(* IEC 61131-3 sources: std_i2980_v2.06_cp053/Source/IMM/ieccontrol/PumpGeneral, 8 files *)

(* ---- ABMeasure.pu ---- *)
(*
@h    ! WARNING !
@h    The Kemro K2 system (including software) only meets category B according to EN 954-1,
@h    thus it is not intended for usage in safety-relevant control applications in the field
@h    of personal safety (e.g. emergency stop).
@h    To implement potentially necessary safety-relevant control tasks, always use additional
@h    external safety devices that are intended for the particular purpose, and meet the necessary
@h    functional safety.
@h    For further information see EN 954-1 (EN ISO 13849-1) and/or the K2-x00 user manual, chapter
@h    "CE conformity, directives and standards".
*)

IMPORT_OVER_LISTFILE
 KAPPL_LintabData_2P
, KAPPL_MeasureMonitoring
, KSWO_Status
, ABMeasureAI

END_IMPORT

ALGORITHM_BLOCK ABMeasure #DUMMY_EDIT_BLOCK

SYSTEM_VAR
 sv_rActPressureHydr : REAL (* actual pressure in bar (measured by pressure sensor) *);
 ai_SysPressure : REAL;
 sv_SysPressureLintab : KAPPL_LintabData_2P (* lintab for measurement of system pressure sensor *);
 sv_SysPresMonitorMeas : KAPPL_MeasureMonitoring;
 sv_bDeviceReady : BOOL;
END_VAR

SYSTEM_OBJECT
 TaskInject : TASK;
 TaskSlow : TASK;
END_OBJECT

PROCESS_ALGORITHM paInitDebugMeasurement ON TaskSlow AUTOSTART

VAR
 variableName : STRING(255);
 swoState : KSWO_Status;
END_VAR
#BEGIN_EDIT_BLOCK
(**************************************** WARNING ********************************************
 *** The KEBA Kemro K2 System including software is not intended for safety control tasks! ***
 ***                       For further information see Comment tab!                        ***
 *********************************************************************************************)

variableName := CONCAT(GET_MY_FU_NAME(),'.sv_rActPressureHydr');
swoState := KSWO_AddVariable( Task := TaskInject,
                              Name := variableName,
                              Variable := sv_rActPressureHydr);

STOP_PROCESS_ALGORITHM();

;#END_EDIT_BLOCK END_ALGORITHM

PROCESS_ALGORITHM paMeasurePressure ON TaskInject(1000) AUTOSTART

VAR_TEMP
 b : BOOL;
END_VAR

VAR
 abPressureMeasure : ABMeasureAI;
 bSensorLinked : BOOL;
 sEndPoint : STRING(64);
END_VAR

(* IecGraph-Code *)

(* init step *)
INITIAL_STEP S_Start:
ACheckSensor (P);
END_STEP

ACTION ACheckSensor: #BEGIN_EDIT_BLOCK
bSensorLinked := IS_LINKED(ai_SysPressure);

;#END_EDIT_BLOCK END_ACTION (*ACheckSensor*)

(* steps *)
STEP S_Stop:
AStop (P);
END_STEP

ACTION AStop: #BEGIN_EDIT_BLOCK
STOP_PROCESS_ALGORITHM();

;#END_EDIT_BLOCK END_ACTION (*AStop*)
STEP S_Init:
AInitMeasure (P);
END_STEP

STEP S_Measure:
AMeasure (N);
END_STEP

(* transitions *)
TRANSITION TLinked (* TLinked *) FROM S_Start TO S_Init :=  #BEGIN_EDIT_BLOCK
bSensorLinked
;#END_EDIT_BLOCK
END_TRANSITION

TRANSITION TNotLinked (* TNotLinked *) FROM S_Start TO S_Stop :=  #BEGIN_EDIT_BLOCK
NOT bSensorLinked
;#END_EDIT_BLOCK
END_TRANSITION

TRANSITION TStop (* TStop *) FROM S_Stop TO S_Start :=  #BEGIN_EDIT_BLOCK
TRUE
;#END_EDIT_BLOCK
END_TRANSITION

TRANSITION TInitDone (* TInitDone *) FROM S_Init TO S_Measure :=  #BEGIN_EDIT_BLOCK
TRUE
;#END_EDIT_BLOCK
END_TRANSITION

(* end IecGraph-Code *)
(* sfc-code *)

(* stand alone actions *)
ACTION AInitMeasure: #BEGIN_EDIT_BLOCK
(**************************************** WARNING ********************************************
 *** The KEBA Kemro K2 System including software is not intended for safety control tasks! ***
 ***                       For further information see Comment tab!                        ***
 *********************************************************************************************)

sEndPoint := CONCAT(GET_MY_FU_NAME(),".ai_SysPressure");

abPressureMeasure.aInit(sRawValue:= sEndPoint,
                        pLintabPointArray := @sv_SysPressureLintab.LintabPoints.Point,
                        piUsedLintabPoints := @sv_SysPressureLintab.LintabPoints.uNoOfPoints);

abPressureMeasure.aInitMonitoring(bEnable := sv_SysPresMonitorMeas.EnableMonitoring,
                                  rLowLimit := sv_SysPresMonitorMeas.LowerLimit,
                                  bLimitation := sv_SysPresMonitorMeas.Limitation,
                                  rFailureFactor := sv_SysPresMonitorMeas.FailureFactor);

;#END_EDIT_BLOCK END_ACTION (*AInitMeasure*)
ACTION AMeasure: #BEGIN_EDIT_BLOCK
(**************************************** WARNING ********************************************
 *** The KEBA Kemro K2 System including software is not intended for safety control tasks! ***
 ***                       For further information see Comment tab!                        ***
 *********************************************************************************************)

abPressureMeasure.aRunLight(bIdle := sv_bDeviceReady);

b := WRITE_SVREAL_DIRECT(sv_rActPressureHydr, abPressureMeasure.aRunLight.rValue);

;#END_EDIT_BLOCK END_ACTION (*AMeasure*)
(* end sfc-code *)

END_ALGORITHM

END_ALGORITHM_BLOCK

#END_OF_IEC_PART

@Puma @IecEditor 6 149 @Pou 25
@@@BEG_Comment@@@
@h    ! WARNING !
@h    The Kemro K2 system (including software) only meets category B according to EN 954-1,
@h    thus it is not intended for usage in safety-relevant control applications in the field
@h    of personal safety (e.g. emergency stop).
@h    To implement potentially necessary safety-relevant control tasks, always use additional
@h    external safety devices that are intended for the particular purpose, and meet the necessary
@h    functional safety.
@h    For further information see EN 954-1 (EN ISO 13849-1) and/or the K2-x00 user manual, chapter
@h    "CE conformity, directives and standards".
@@@END_Comment@@@

@BEG_Contents

@BEG_Func
@RT(17)FuncTreeContainer
0
@END_Func

@BEG_Const
@RT(18)ConstTreeContainer
0
@END_Const

@BEG_Export

@BEG_Kind
@ALGORITHM_BLOCK @RT(9)ABMeasure @STRUCTURED_TEXT
@RT(0) @RT(0) @RT(0)
@END_Kind

@BEG_Dcl
@RT(16)DclTreeContainer
7
@Var @RT(10)TaskInject @RT(0) @T @T @RENAMED 0 @T @T @DT @RT(4)TASK @RT(0) @T @T @BASIC 0 @F
@F @F
@T
@BEG_Attrib
3 @RT(0) @RT(0) @RT(0)
@END_Attrib
1 7 @F @F @F @F

@Var @RT(8)TaskSlow @RT(0) @T @T @RENAMED 0 @T @T @DT @RT(4)TASK @RT(0) @T @T @BASIC 0 @F
@F @F
@T
@BEG_Attrib
3 @RT(0) @RT(0) @RT(0)
@END_Attrib
1 7 @F @F @F @F

@Var @RT(19)sv_rActPressureHydr @RT(0) @T @F @DT @RT(4)REAL @RT(0) @T @T @BASIC 0 @F
@F @F
@T
@BEG_Attrib
3 @RT(0) @RT(52)actual pressure in bar (measured by pressure sensor) @RT(0)
@END_Attrib
1 8 @F @F @F @F

@Var @RT(14)ai_SysPressure @RT(0) @T @F @DT @RT(4)REAL @RT(0) @T @T @BASIC 0 @F
@F @F
@T
@BEG_Attrib
3 @RT(0) @RT(0) @RT(0)
@END_Attrib
1 8 @F @F @F @F

@Var @RT(20)sv_SysPressureLintab @RT(0) @T @T @DERIVED 0 @F @RT(19)KAPPL_LintabData_2P @F
@T
@BEG_Attrib
3 @RT(0) @RT(48)lintab for measurement of system pressure sensor @RT(0)
@END_Attrib
1 8 @F @F @F @F

@Var @RT(21)sv_SysPresMonitorMeas @RT(0) @T @T @DERIVED 0 @T @T @DT @RT(23)KAPPL_MeasureMonitoring @RT(0) @T @T @UNKNOWN 0 @F
@F @F
@T
@BEG_Attrib
3 @RT(0) @RT(0) @RT(0)
@END_Attrib
1 8 @F @F @F @F

@Var @RT(15)sv_bDeviceReady @RT(0) @T @F @DT @RT(4)BOOL @RT(0) @T @T @BASIC 0 @F
@F @F
@T
@BEG_Attrib
3 @RT(0) @RT(0) @RT(0)
@END_Attrib
1 8 @F @F @F @F

@END_Dcl

@END_Export

@BEG_Body

2

@BEG_Export

@BEG_Algo
@PROCESS_ALGORITHM @RT(22)paInitDebugMeasurement @STRUCTURED_TEXT
@RT(0) @RT(0) @RT(8)TaskSlow @T @F
@END_Algo

@BEG_Dcl
@RT(16)DclTreeContainer
2
@Var @RT(12)variableName @RT(0) @T @F @DT @RT(11)STRING(255) @RT(0) @T @T @STRING 0 @F @RT(3)255 @F
@F @F
@T
@BEG_Attrib
3 @RT(0) @RT(0) @RT(0)
@END_Attrib
1 0 @F @F @F @F

@Var @RT(8)swoState @RT(0) @T @T @DERIVED 0 @T @T @DT @RT(11)KSWO_Status @RT(0) @T @T @UNKNOWN 0 @F
@F @F
@T
@BEG_Attrib
3 @RT(0) @RT(0) @RT(0)
@END_Attrib
1 0 @F @F @F @F

@END_Dcl

@END_Export

@BEG_Export

@BEG_Algo
@PROCESS_ALGORITHM @RT(17)paMeasurePressure @SEQUENTIAL_FLOW_CHART
@RT(0) @RT(0) @RT(16)TaskInject(1000) @T @F
@END_Algo

@BEG_Dcl
@RT(16)DclTreeContainer
4
@Var @RT(17)abPressureMeasure @RT(0) @T @T @DERIVED 0 @F @RT(11)ABMeasureAI @F
@T
@BEG_Attrib
3 @RT(0) @RT(0) @RT(0)
@END_Attrib
1 0 @F @F @F @F

@Var @RT(13)bSensorLinked @RT(0) @T @F @DT @RT(4)BOOL @RT(0) @T @T @BASIC 0 @F
@F @F
@T
@BEG_Attrib
3 @RT(0) @RT(0) @RT(0)
@END_Attrib
1 0 @F @F @F @F

@Var @RT(9)sEndPoint @RT(0) @T @F @DT @RT(10)STRING(64) @RT(0) @T @T @STRING 0 @F @RT(2)64 @F
@F @F
@T
@BEG_Attrib
3 @RT(0) @RT(0) @RT(0)
@END_Attrib
1 0 @F @F @F @F

@Var @RT(1)b @RT(0) @T @F @DT @RT(4)BOOL @RT(0) @T @T @BASIC 0 @F
@F @F
@T
@BEG_Attrib
3 @RT(0) @RT(0) @RT(0)
@END_Attrib
1 4 @F @F @F @F

@END_Dcl

@END_Export

@BEG_Body
@TL(12)
(**************************************** WARNING ********************************************
 *** The KEBA Kemro K2 System including software is not intended for safety control tasks! ***
 ***                       For further information see Comment tab!                        ***
 *********************************************************************************************)

variableName := CONCAT(GET_MY_FU_NAME(),'.sv_rActPressureHydr');
swoState := KSWO_AddVariable( Task := TaskInject,
                              Name := variableName,
                              Variable := sv_rActPressureHydr);

STOP_PROCESS_ALGORITHM();

@END_Body

@@@BEG_Comment@@@
@TL(0)

@@@END_Comment@@@

@BEG_SfcBody
8 6 5

@BEG_SfcData 2
@StepSeq @RT(4)sseq @F 5
@Step @RT(7)S_Start @F @T @T @F @RT(0) @F
@AcbCont @RT(7)unnamed @F 1
@Acb @RT(12)ACheckSensor @F @T @RT(1)P @RT(0) @F @F @T @TL(2)
bSensorLinked := IS_LINKED(ai_SysPressure);

@F

@AltBranch @RT(3)alt @F 2
@TransSeq @RT(4)tseq @F 1
@Trans @RT(7)TLinked @F @T @F @F @T @T @TL(2)
bSensorLinked

@RT(7)TLinked @F

@TransSeq @RT(4)tseq @F 4
@Trans @RT(10)TNotLinked @F @T @F @F @T @T @TL(2)
NOT bSensorLinked

@RT(10)TNotLinked @F
@Step @RT(6)S_Stop @F @F @F @F @RT(0) @F
@AcbCont @RT(7)unnamed @F 1
@Acb @RT(5)AStop @F @T @RT(1)P @RT(0) @F @F @T @TL(2)
STOP_PROCESS_ALGORITHM();

@F

@Trans @RT(5)TStop @F @T @F @F @T @T @TL(2)
TRUE

@RT(5)TStop @F
@Goto @RT(7)S_Start @F @F

@Step @RT(6)S_Init @F @F @F @F @RT(0) @F
@AcbCont @RT(7)unnamed @F 1
@Acb @RT(12)AInitMeasure @F @F @RT(1)P @RT(0) @F @F @F @F

@Trans @RT(9)TInitDone @F @T @F @F @T @T @TL(2)
TRUE

@RT(9)TInitDone @F
@Step @RT(9)S_Measure @F @F @F @F @RT(0) @F
@AcbCont @RT(7)unnamed @F 1
@Acb @RT(8)AMeasure @F @F @RT(1)N @RT(0) @F @F @F @F

@END_SfcData
@SaActions 2
@SaText @RT(12)AInitMeasure 1 @TL(17)
(**************************************** WARNING ********************************************
 *** The KEBA Kemro K2 System including software is not intended for safety control tasks! ***
 ***                       For further information see Comment tab!                        ***
 *********************************************************************************************)

sEndPoint := CONCAT(GET_MY_FU_NAME(),".ai_SysPressure");

abPressureMeasure.aInit(sRawValue:= sEndPoint,
                        pLintabPointArray := @sv_SysPressureLintab.LintabPoints.Point,
                        piUsedLintabPoints := @sv_SysPressureLintab.LintabPoints.uNoOfPoints);

abPressureMeasure.aInitMonitoring(bEnable := sv_SysPresMonitorMeas.EnableMonitoring,
                                  rLowLimit := sv_SysPresMonitorMeas.LowerLimit,
                                  bLimitation := sv_SysPresMonitorMeas.Limitation,
                                  rFailureFactor := sv_SysPresMonitorMeas.FailureFactor);

@SaText @RT(8)AMeasure 1 @TL(9)
(**************************************** WARNING ********************************************
 *** The KEBA Kemro K2 System including software is not intended for safety control tasks! ***
 ***                       For further information see Comment tab!                        ***
 *********************************************************************************************)

abPressureMeasure.aRunLight(bIdle := sv_bDeviceReady);

b := WRITE_SVREAL_DIRECT(sv_rActPressureHydr, abPressureMeasure.aRunLight.rValue);

@SaTrans 0
@SaExits 0
@END_SfcBody

@@@BEG_Comment@@@
@TL(0)

@@@END_Comment@@@
@END_Body

@END_Contents

(* ---- ABOutSpeedPump.pu ---- *)
(*
ATTENTION: Task for paOut is maybe mapped to another task because Inject and Mold run with 1ms
*)

IMPORT_OVER_LISTFILE
 WRITE_SVREAL_DIRECT
, cMoveAll
, nLockAbort
, cMaxDeviceMovements
, cMoveNone
, nUnlock
, nOperationState_AF
, tsTraceLevel
, tsServo
, KHW_Servo_Data
, FBDebugTrace
, tsPQForce

END_IMPORT

ALGORITHM_BLOCK ABOutSpeedPump #DUMMY_EDIT_BLOCK

SYSTEM_VAR
 sv_TraceLevel : tsTraceLevel;
 sv_Servo : tsServo;
 sv_bInitDone : BOOL;
 sv_bEmergencyStop : BOOL;
 sv_KHW_Servo_setValue : KHW_Servo_Data;
 sv_ForceP : tsPQForce (* pressure force  *);
 sv_ForceQ : tsPQForce (* flow force *);
 sv_rDrivePressure : REAL;
 sv_rDriveVelocity : REAL;
END_VAR

SYSTEM_OBJECT
 TaskMid : TASK;
 TaskAnalog : TASK (* ATTENTION: MAYBE MAPPED *);
 PU_Task_7 : TASK;
END_OBJECT

VAR
 fbDebugTrace : FBDebugTrace;
 mbInitDone : BOOL;
 mbStop : BOOL;
 mbDriveError : BOOL;
 mbForceStarted : BOOL;
END_VAR

PROCESS_ALGORITHM paInit ON TaskMid AUTOSTART

VAR
 bInit : BOOL;
END_VAR
#BEGIN_EDIT_BLOCK
(**************************************** WARNING ********************************************
 *** The KEBA Kemro K2 System including software is not intended for safety control tasks! ***
 ***                       For further information see Comment tab!                        ***
 *********************************************************************************************)
IF NOT IS_LINKED(sv_KHW_Servo_setValue) THEN
    RETURN;
END_IF;

IF NOT bInit AND sv_bInitDone THEN

   bInit := TRUE;
   IF NOT IS_LINKED(sv_Servo) THEN
      IF sv_TraceLevel.bAnalog THEN
         fbDebugTrace.sText := 'ABOutSpeedPump.paInit: sv_Servo not linked';
         fbDebugTrace();
      END_IF;
   END_IF;
END_IF;

IF bInit THEN
   // all required data for analog output are ok -> start DriveInit
   IF sv_Servo.bInitDone THEN
      mbInitDone := TRUE;
      STOP_PROCESS_ALGORITHM();
   ELSE
      sv_Servo.bInitStart := TRUE;
   END_IF;
ELSIF sv_bInitDone THEN
   STOP_PROCESS_ALGORITHM();
END_IF;

;#END_EDIT_BLOCK END_ALGORITHM

PROCESS_ALGORITHM paOut ON TaskAnalog(15001)

VAR_TEMP
 b : BOOL;
END_VAR

(* IecGraph-Code *)

(* init step *)
INITIAL_STEP INIT:
END_STEP

(* steps *)
STEP OUT:
aOut (N);
END_STEP

STEP IDLE_OUT:
aStopOut (P);
END_STEP

STEP STOP:
aStopOut (P);
Action3 (P);
END_STEP

ACTION Action3: #BEGIN_EDIT_BLOCK
IF mbStop OR mbDriveError OR sv_bEmergencyStop THEN
   STOP_PROCESS_ALGORITHM();
END_IF;

;#END_EDIT_BLOCK END_ACTION (*Action3*)

(* transitions *)
GO_ON_TRANSITION Trans1 (* Trans1 *) FROM INIT TO OUT :=  #BEGIN_EDIT_BLOCK
sv_Servo.ServoState.OperationState
= nOperationState_AF

;#END_EDIT_BLOCK
END_TRANSITION

TRANSITION Trans13 (* Trans13 *) FROM INIT TO STOP :=  #BEGIN_EDIT_BLOCK
mbStop OR
mbDriveError OR
sv_bEmergencyStop

;#END_EDIT_BLOCK
END_TRANSITION

GO_ON_TRANSITION Trans2 (* Trans2 *) FROM OUT TO STOP :=  #BEGIN_EDIT_BLOCK
mbStop OR mbDriveError OR
sv_bEmergencyStop
;#END_EDIT_BLOCK
(*Use GoOn transitions to avoid timing problem
between releasing and requesting the drive!*)
END_TRANSITION

GO_ON_TRANSITION Trans4 (* Trans4 *) FROM OUT TO IDLE_OUT :=  #BEGIN_EDIT_BLOCK
sv_Servo.ServoState.OperationState
<> nOperationState_AF
;#END_EDIT_BLOCK
END_TRANSITION

TRANSITION Trans6 (* Trans6 *) FROM IDLE_OUT TO OUT :=  #BEGIN_EDIT_BLOCK
sv_Servo.ServoState.OperationState
= nOperationState_AF
;#END_EDIT_BLOCK
END_TRANSITION

GO_ON_TRANSITION Trans7 (* Trans7 *) FROM IDLE_OUT TO STOP :=  #BEGIN_EDIT_BLOCK
mbStop OR mbDriveError
;#END_EDIT_BLOCK
END_TRANSITION

TRANSITION Trans3 (* Trans3 *) FROM STOP TO INIT :=  #BEGIN_EDIT_BLOCK
TRUE
;#END_EDIT_BLOCK
END_TRANSITION

(* end IecGraph-Code *)
(* sfc-code *)

(* stand alone actions *)
ACTION aStopOut: #BEGIN_EDIT_BLOCK

sv_KHW_Servo_setValue.rVeloc := 0.0;
sv_KHW_Servo_setValue.rAux[2] := 0.0;

;#END_EDIT_BLOCK END_ACTION (*aStopOut*)
ACTION aOut: #BEGIN_EDIT_BLOCK
//Assignment PQ endpoints
b := WRITE_SVREAL_DIRECT(sv_KHW_Servo_setValue.rAux[1], sv_rDrivePressure);
b := WRITE_SVREAL_DIRECT(sv_KHW_Servo_setValue.rVeloc, sv_rDriveVelocity);

;#END_EDIT_BLOCK END_ACTION (*aOut*)
(* end sfc-code *)

END_ALGORITHM

ALGORITHM aStart

VAR_INPUT
 piCtrlParamSet : REFTO INT;
 bMaster : BOOL (* TRUE: pump is master, FALSE: pump is slave *);
END_VAR

VAR_TEMP
 b : BOOL;
END_VAR

VAR
 rTmp : REAL;
END_VAR
#BEGIN_EDIT_BLOCK
(**************************************** WARNING ********************************************
 *** The KEBA Kemro K2 System including software is not intended for safety control tasks! ***
 ***                       For further information see Comment tab!                        ***
 *********************************************************************************************)

IF mbInitDone THEN

   IF NOT sv_Servo.ServoState.bError THEN

      //Bit 0: first or second parameter set (first parameter set should be default)
      //Bit 1: master or slave (master = 0, slave = 1)
      IF bMaster THEN
         rTmp := 0.0;
      ELSE
         rTmp := 2.0;
      END_IF;

      IF CHECK_REF(piCtrlParamSet^) AND (piCtrlParamSet^ = 2) THEN
         rTmp := rTmp + 1.0;
      END_IF;

      b := WRITE_SV_DIRECT(sv_KHW_Servo_setValue.rAux[2], rTmp);

      mbStop := FALSE;
      START_PROCESS_ALGORITHM(paOut);

    END_IF;
END_IF;

;#END_EDIT_BLOCK END_ALGORITHM

ALGORITHM aStop

#BEGIN_EDIT_BLOCK
(**************************************** WARNING ********************************************
 *** The KEBA Kemro K2 System including software is not intended for safety control tasks! ***
 ***                       For further information see Comment tab!                        ***
 *********************************************************************************************)

mbStop := TRUE;

;#END_EDIT_BLOCK END_ALGORITHM

POSTUPDATE_ALGORITHM pDriveError ON PU_Task_7 WITH sv_Servo.ServoState.bError,sv_Servo.bInitDone

#BEGIN_EDIT_BLOCK
(**************************************** WARNING ********************************************
 *** The KEBA Kemro K2 System including software is not intended for safety control tasks! ***
 ***                       For further information see Comment tab!                        ***
 *********************************************************************************************)

IF NOT IS_LINKED(sv_KHW_Servo_setValue) THEN
   RETURN;
END_IF;

mbDriveError := sv_Servo.ServoState.bError;

;#END_EDIT_BLOCK END_ALGORITHM

POSTUPDATE_ALGORITHM pPQForce ON PU_Task_7 WITH sv_ForceP.bForce,sv_ForceQ.bForce

#BEGIN_EDIT_BLOCK
(**************************************** WARNING ********************************************
 *** The KEBA Kemro K2 System including software is not intended for safety control tasks! ***
 ***                       For further information see Comment tab!                        ***
 *********************************************************************************************)

//Force PQ endpoints
IF sv_ForceP.bForce OR sv_ForceQ.bForce THEN
   IF NOT mbForceStarted THEN
      mbForceStarted := TRUE;
      START_PROCESS_ALGORITHM(paPQForce);
   END_IF;
END_IF;

;#END_EDIT_BLOCK END_ALGORITHM

PROCESS_ALGORITHM paPQForce ON TaskAnalog

VAR_TEMP
 rForceP : REAL;
 rForceQ : REAL;
 b : BOOL;
END_VAR

VAR CONSTANT
 rMaxPressure : REAL := 400.0;
END_VAR
#BEGIN_EDIT_BLOCK
(**************************************** WARNING ********************************************
 *** The KEBA Kemro K2 System including software is not intended for safety control tasks! ***
 ***                       For further information see Comment tab!                        ***
 *********************************************************************************************)

//Force PQ endpoints
IF sv_ForceP.bForce THEN
   rForceP := sv_ForceP.rForceValue / rMaxPressure * 1000.0;
   b := WRITE_SVREAL_DIRECT(sv_KHW_Servo_setValue.rAux[1], rForceP);
   b := WRITE_SVREAL_DIRECT(sv_ForceP.rActualValue, sv_ForceP.rForceValue);
ELSIF NOT sv_ForceP.bForce THEN
   b := WRITE_SVREAL_DIRECT(sv_KHW_Servo_setValue.rAux[1], 0.0);
   b := WRITE_SVREAL_DIRECT(sv_ForceP.rActualValue, 0.0);
END_IF;

IF sv_ForceQ.bForce THEN
   rForceQ := sv_ForceQ.rForceValue * 10.0;
   b := WRITE_SVREAL_DIRECT(sv_KHW_Servo_setValue.rVeloc, rForceQ);
   b := WRITE_SVREAL_DIRECT(sv_ForceQ.rActualValue, sv_ForceQ.rForceValue);
ELSIF NOT sv_ForceQ.bForce THEN
   b := WRITE_SVREAL_DIRECT(sv_KHW_Servo_setValue.rVeloc, 0.0);
   b := WRITE_SVREAL_DIRECT(sv_ForceQ.rActualValue, 0.0);
END_IF;

IF NOT sv_ForceQ.bForce AND NOT sv_ForceP.bForce THEN
   mbForceStarted := FALSE;
   STOP_PROCESS_ALGORITHM();
END_IF;

;#END_EDIT_BLOCK END_ALGORITHM

END_ALGORITHM_BLOCK

#END_OF_IEC_PART

@Puma @IecEditor 6 114 @Pou 25
@@@BEG_Comment@@@
ATTENTION: Task for paOut is maybe mapped to another task because Inject and Mold run with 1ms
@@@END_Comment@@@

@BEG_Contents

@BEG_Func
@RT(17)FuncTreeContainer
1
@Var @RT(19)WRITE_SVREAL_DIRECT @RT(0) @T @T @DERIVED 0 @F @RT(22)KEBA_STANDARD_FUNCTION @F
@T
@BEG_Attrib
0 @RT(0) @RT(0)
@END_Attrib
1 1 @F @F @F @F

@END_Func

@BEG_Const
@RT(18)ConstTreeContainer
6
@Var @RT(8)cMoveAll @RT(0) @T @F @DT @RT(4)DINT @RT(0) @T @T @BASIC 0 @F
@F @F
@T
@BEG_Attrib
0 @RT(13)cMaxMoveIdent @RT(32)all movements (for evLockUnlock)
@END_Attrib
1 1 @F @F @F @F

@Var @RT(10)nLockAbort @RT(0) @T @T @DERIVED 0 @F @RT(12)tnLockUnlock @F
@T
@BEG_Attrib
0 @RT(1)0 @RT(0)
@END_Attrib
1 1 @F @F @F @F

@Var @RT(19)cMaxDeviceMovements @RT(0) @T @F @DT @RT(4)DINT @RT(0) @T @T @BASIC 0 @F
@F @F
@T
@BEG_Attrib
0 @RT(2)20 @RT(34)max number of movements per device
@END_Attrib
1 1 @F @F @F @F

@Var @RT(9)cMoveNone @RT(0) @T @F @DT @RT(4)DINT @RT(0) @T @T @BASIC 0 @F
@F @F
@T
@BEG_Attrib
0 @RT(13)cMinMoveIdent @RT(4)None
@END_Attrib
1 1 @F @F @F @F

@Var @RT(7)nUnlock @RT(0) @T @T @DERIVED 0 @F @RT(12)tnLockUnlock @F
@T
@BEG_Attrib
0 @RT(1)2 @RT(0)
@END_Attrib
1 1 @F @F @F @F

@Var @RT(18)nOperationState_AF @RT(0) @T @T @DERIVED 0 @F @RT(16)tnOperationState @F
@T
@BEG_Attrib
0 @RT(1)4 @RT(12)drive enable
@END_Attrib
1 1 @F @F @F @F

@END_Const

@BEG_Export

@BEG_Kind
@ALGORITHM_BLOCK @RT(14)ABOutSpeedPump @STRUCTURED_TEXT
@RT(0) @RT(0) @RT(0)
@END_Kind

@BEG_Dcl
@RT(16)DclTreeContainer
17
@Var @RT(13)sv_TraceLevel @RT(0) @T @T @DERIVED 0 @T @T @DT @RT(12)tsTraceLevel @RT(0) @T @T @UNKNOWN 0 @F
@F @F
@T
@BEG_Attrib
3 @RT(0) @RT(0) @RT(0)
@END_Attrib
1 8 @F @F @F @F

@Var @RT(8)sv_Servo @RT(0) @T @T @DERIVED 0 @T @T @DT @RT(7)tsServo @RT(0) @T @T @UNKNOWN 0 @F
@F @F
@T
@BEG_Attrib
3 @RT(0) @RT(0) @RT(0)
@END_Attrib
1 8 @F @F @F @F

@Var @RT(12)sv_bInitDone @RT(0) @T @F @DT @RT(4)BOOL @RT(0) @T @T @BASIC 0 @F
@F @F
@T
@BEG_Attrib
3 @RT(0) @RT(0) @RT(0)
@END_Attrib
1 8 @F @F @F @F

@Var @RT(17)sv_bEmergencyStop @RT(0) @T @F @DT @RT(4)BOOL @RT(0) @T @T @BASIC 0 @F
@F @F
@T
@BEG_Attrib
3 @RT(0) @RT(0) @RT(0)
@END_Attrib
1 8 @F @F @F @F

@Var @RT(21)sv_KHW_Servo_setValue @RT(0) @T @T @DERIVED 0 @T @T @DT @RT(14)KHW_Servo_Data @RT(0) @T @T @UNKNOWN 0 @F
@F @F
@T
@BEG_Attrib
3 @RT(0) @RT(0) @RT(0)
@END_Attrib
1 8 @F @F @F @F

@Var @RT(7)TaskMid @RT(0) @T @F @DT @RT(4)TASK @RT(0) @T @T @BASIC 0 @F
@F @F
@T
@BEG_Attrib
3 @RT(0) @RT(0) @RT(0)
@END_Attrib
1 7 @F @F @F @F

@Var @RT(10)TaskAnalog @RT(0) @T @F @DT @RT(4)TASK @RT(0) @T @T @BASIC 0 @F
@F @F
@T
@BEG_Attrib
3 @RT(0) @RT(23)ATTENTION: MAYBE MAPPED @RT(0)
@END_Attrib
1 7 @F @F @F @F

@Var @RT(9)PU_Task_7 @RT(0) @T @F @DT @RT(4)TASK @RT(0) @T @T @BASIC 0 @F
@F @F
@T
@BEG_Attrib
3 @RT(0) @RT(0) @RT(0)
@END_Attrib
1 7 @F @F @F @F

@Var @RT(12)fbDebugTrace @RT(0) @T @T @DERIVED 0 @T @T @DT @RT(12)FBDebugTrace @RT(0) @T @T @UNKNOWN 0 @F
@F @F
@T
@BEG_Attrib
3 @RT(0) @RT(0) @RT(0)
@END_Attrib
1 0 @F @F @F @F

@Var @RT(10)mbInitDone @RT(0) @T @F @DT @RT(4)BOOL @RT(0) @T @T @BASIC 0 @F
@F @F
@T
@BEG_Attrib
3 @RT(0) @RT(0) @RT(0)
@END_Attrib
1 0 @F @F @F @F

@Var @RT(6)mbStop @RT(0) @T @F @DT @RT(4)BOOL @RT(0) @T @T @BASIC 0 @F
@F @F
@T
@BEG_Attrib
3 @RT(0) @RT(0) @RT(0)
@END_Attrib
1 0 @F @F @F @F

@Var @RT(12)mbDriveError @RT(0) @T @F @DT @RT(4)BOOL @RT(0) @T @T @BASIC 0 @F
@F @F
@T
@BEG_Attrib
3 @RT(0) @RT(0) @RT(0)
@END_Attrib
1 0 @F @F @F @F

@Var @RT(9)sv_ForceP @RT(0) @T @T @DERIVED 0 @T @T @DT @RT(9)tsPQForce @RT(0) @T @T @UNKNOWN 0 @F
@F @F
@T
@BEG_Attrib
3 @RT(0) @RT(15)pressure force  @RT(0)
@END_Attrib
1 8 @F @F @F @F

@Var @RT(9)sv_ForceQ @RT(0) @T @T @DERIVED 0 @T @T @DT @RT(9)tsPQForce @RT(0) @T @T @UNKNOWN 0 @F
@F @F
@T
@BEG_Attrib
3 @RT(0) @RT(10)flow force @RT(0)
@END_Attrib
1 8 @F @F @F @F

@Var @RT(14)mbForceStarted @RT(0) @T @T @RENAMED 0 @T @T @DT @RT(4)BOOL @RT(0) @T @T @BASIC 0 @F
@F @F
@T
@BEG_Attrib
3 @RT(0) @RT(0) @RT(0)
@END_Attrib
1 0 @F @F @F @F

@Var @RT(17)sv_rDrivePressure @RT(0) @T @F @DT @RT(4)REAL @RT(0) @T @T @BASIC 0 @F
@F @F
@T
@BEG_Attrib
3 @RT(0) @RT(0) @RT(0)
@END_Attrib
1 8 @F @F @F @F

@Var @RT(17)sv_rDriveVelocity @RT(0) @T @F @DT @RT(4)REAL @RT(0) @T @T @BASIC 0 @F
@F @F
@T
@BEG_Attrib
3 @RT(0) @RT(0) @RT(0)
@END_Attrib
1 8 @F @F @F @F

@END_Dcl

@END_Export

@BEG_Body

7

@BEG_Export

@BEG_Algo
@PROCESS_ALGORITHM @RT(6)paInit @STRUCTURED_TEXT
@RT(0) @RT(0) @RT(7)TaskMid @T @F
@END_Algo

@BEG_Dcl
@RT(16)DclTreeContainer
1
@Var @RT(5)bInit @RT(0) @T @F @DT @RT(4)BOOL @RT(0) @T @T @BASIC 0 @F
@F @F
@T
@BEG_Attrib
3 @RT(0) @RT(0) @RT(0)
@END_Attrib
1 0 @F @F @F @F

@END_Dcl

@END_Export

@BEG_Export

@BEG_Algo
@PROCESS_ALGORITHM @RT(5)paOut @SEQUENTIAL_FLOW_CHART
@RT(0) @RT(0) @RT(17)TaskAnalog(15001) @F @F
@END_Algo

@BEG_Dcl
@RT(16)DclTreeContainer
1
@Var @RT(1)b @RT(0) @T @F @DT @RT(4)BOOL @RT(0) @T @T @BASIC 0 @F
@F @F
@T
@BEG_Attrib
3 @RT(0) @RT(0) @RT(0)
@END_Attrib
1 4 @F @F @F @F

@END_Dcl

@END_Export

@BEG_Export

@BEG_Algo
@ALGORITHM @RT(6)aStart @STRUCTURED_TEXT
@RT(0) @RT(0) @RT(0) @F @F
@END_Algo

@BEG_Dcl
@RT(16)DclTreeContainer
4
@Var @RT(14)piCtrlParamSet @RT(0) @T @T @REFTO 0 @T @DT @RT(3)INT @RT(0) @T @T @BASIC 0 @F
@F @F
@T
@BEG_Attrib
3 @RT(0) @RT(0) @RT(0)
@END_Attrib
1 1 @F @F @F @F

@Var @RT(7)bMaster @RT(0) @T @F @DT @RT(4)BOOL @RT(0) @T @T @BASIC 0 @F
@F @F
@T
@BEG_Attrib
3 @RT(0) @RT(42)TRUE: pump is master, FALSE: pump is slave @RT(0)
@END_Attrib
1 1 @F @F @F @F

@Var @RT(4)rTmp @RT(0) @T @F @DT @RT(4)REAL @RT(0) @T @T @BASIC 0 @F
@F @F
@T
@BEG_Attrib
3 @RT(0) @RT(0) @RT(0)
@END_Attrib
1 0 @F @F @F @F

@Var @RT(1)b @RT(0) @T @F @DT @RT(4)BOOL @RT(0) @T @T @BASIC 0 @F
@F @F
@T
@BEG_Attrib
3 @RT(0) @RT(0) @RT(0)
@END_Attrib
1 4 @F @F @F @F

@END_Dcl

@END_Export

@BEG_Export

@BEG_Algo
@ALGORITHM @RT(5)aStop @STRUCTURED_TEXT
@RT(0) @RT(0) @RT(0) @F @F
@END_Algo

@BEG_Dcl
@RT(16)DclTreeContainer
0
@END_Dcl

@END_Export

@BEG_Export

@BEG_Algo
@POSTUPDATE_ALGORITHM @RT(11)pDriveError @STRUCTURED_TEXT
@RT(0) @RT(45)sv_Servo.ServoState.bError,sv_Servo.bInitDone @RT(9)PU_Task_7 @F @F
@END_Algo

@BEG_Dcl
@RT(16)DclTreeContainer
0
@END_Dcl

@END_Export

@BEG_Export

@BEG_Algo
@POSTUPDATE_ALGORITHM @RT(8)pPQForce @STRUCTURED_TEXT
@RT(0) @RT(33)sv_ForceP.bForce,sv_ForceQ.bForce @RT(9)PU_Task_7 @F @F
@END_Algo

@BEG_Dcl
@RT(16)DclTreeContainer
0
@END_Dcl

@END_Export

@BEG_Export

@BEG_Algo
@PROCESS_ALGORITHM @RT(9)paPQForce @STRUCTURED_TEXT
@RT(0) @RT(0) @RT(10)TaskAnalog @F @F
@END_Algo

@BEG_Dcl
@RT(16)DclTreeContainer
4
@Var @RT(12)rMaxPressure @RT(0) @T @F @DT @RT(4)REAL @RT(0) @T @T @BASIC 0 @F
@F @F
@T
@BEG_Attrib
3 @RT(5)400.0 @RT(0) @RT(0)
@END_Attrib
1 15 @F @F @F @F

@Var @RT(7)rForceP @RT(0) @T @F @DT @RT(4)REAL @RT(0) @T @T @BASIC 0 @F
@F @F
@T
@BEG_Attrib
3 @RT(0) @RT(0) @RT(0)
@END_Attrib
1 4 @F @F @F @F

@Var @RT(7)rForceQ @RT(0) @T @F @DT @RT(4)REAL @RT(0) @T @T @BASIC 0 @F
@F @F
@T
@BEG_Attrib
3 @RT(0) @RT(0) @RT(0)
@END_Attrib
1 4 @F @F @F @F

@Var @RT(1)b @RT(0) @T @F @DT @RT(4)BOOL @RT(0) @T @T @BASIC 0 @F
@F @F
@T
@BEG_Attrib
3 @RT(0) @RT(0) @RT(0)
@END_Attrib
1 4 @F @F @F @F

@END_Dcl

@END_Export

@BEG_Body
@TL(32)
(**************************************** WARNING ********************************************
 *** The KEBA Kemro K2 System including software is not intended for safety control tasks! ***
 ***                       For further information see Comment tab!                        ***
 *********************************************************************************************)
IF NOT IS_LINKED(sv_KHW_Servo_setValue) THEN
    RETURN;
END_IF;

IF NOT bInit AND sv_bInitDone THEN

   bInit := TRUE;
   IF NOT IS_LINKED(sv_Servo) THEN
      IF sv_TraceLevel.bAnalog THEN
         fbDebugTrace.sText := 'ABOutSpeedPump.paInit: sv_Servo not linked';
         fbDebugTrace();
      END_IF;
   END_IF;
END_IF;

IF bInit THEN
   // all required data for analog output are ok -> start DriveInit
   IF sv_Servo.bInitDone THEN
      mbInitDone := TRUE;
      STOP_PROCESS_ALGORITHM();
   ELSE
      sv_Servo.bInitStart := TRUE;
   END_IF;
ELSIF sv_bInitDone THEN
   STOP_PROCESS_ALGORITHM();
END_IF;

@END_Body

@@@BEG_Comment@@@
@TL(0)

@@@END_Comment@@@

@BEG_SfcBody
6 8 8

@BEG_SfcData 2
@StepSeq @RT(4)sseq @F 1
@Loop @RT(4)loop @F 2
@StepSeq @RT(4)sseq @F 5
@Step @RT(4)INIT @F @T @F @F @RT(0) @F
@AcbCont @RT(7)unnamed @F 0

@AltBranch @RT(3)alt @F 2
@TransSeq @RT(4)tseq @F 1
@Trans @RT(6)Trans1 @F @T @F @F @T @F @TL(4)
sv_Servo.ServoState.OperationState
= nOperationState_AF

@RT(6)Trans1 @F

@TransSeq @RT(4)tseq @F 2
@Trans @RT(7)Trans13 @F @T @F @F @T @T @TL(5)
mbStop OR
mbDriveError OR
sv_bEmergencyStop

@RT(7)Trans13 @F
@Goto @RT(4)STOP @F @F

@Step @RT(3)OUT @F @F @T @F @RT(0) @F
@AcbCont @RT(7)unnamed @F 1
@Acb @RT(4)aOut @F @F @RT(1)N @RT(0) @F @F @F @F

@AltBranch @RT(3)alt @F 2
@TransSeq @RT(4)tseq @F 1
@Trans @RT(6)Trans2 @F @T @F @F @T @F @TL(3)
mbStop OR mbDriveError OR
sv_bEmergencyStop

@RT(6)Trans2 @T @TL(2)
Use GoOn transitions to avoid timing problem
between releasing and requesting the drive!

@TransSeq @RT(4)tseq @F 4
@Trans @RT(6)Trans4 @F @T @F @F @T @F @TL(3)
sv_Servo.ServoState.OperationState
<> nOperationState_AF

@RT(6)Trans4 @F
@Step @RT(8)IDLE_OUT @F @F @F @F @RT(0) @F
@AcbCont @RT(7)unnamed @F 1
@Acb @RT(8)aStopOut @F @F @RT(1)P @RT(0) @F @F @F @F

@AltBranch @RT(3)alt @F 2
@TransSeq @RT(4)tseq @F 1
@Trans @RT(6)Trans6 @F @T @F @F @T @T @TL(3)
sv_Servo.ServoState.OperationState
= nOperationState_AF

@RT(6)Trans6 @F

@TransSeq @RT(4)tseq @F 2
@Trans @RT(6)Trans7 @F @T @F @F @T @F @TL(2)
mbStop OR mbDriveError

@RT(6)Trans7 @F
@Goto @RT(4)STOP @F @F

@Goto @RT(3)OUT @F @F

@Step @RT(4)STOP @F @F @T @F @RT(0) @F
@AcbCont @RT(7)unnamed @F 2
@Acb @RT(8)aStopOut @F @F @RT(1)P @RT(0) @F @F @F @F
@Acb @RT(7)Action3 @F @T @RT(1)P @RT(0) @F @F @T @TL(4)
IF mbStop OR mbDriveError OR sv_bEmergencyStop THEN
   STOP_PROCESS_ALGORITHM();
END_IF;

@F

@Trans @RT(6)Trans3 @F @T @T @T @T @T @TL(2)
TRUE

@RT(6)Trans3 @F

@END_SfcData
@SaActions 2
@SaText @RT(8)aStopOut 1 @TL(6)

sv_KHW_Servo_setValue.rVeloc := 0.0;
sv_KHW_Servo_setValue.rAux[2] := 0.0;

@SaText @RT(4)aOut 1 @TL(8)
//Assignment PQ endpoints
b := WRITE_SVREAL_DIRECT(sv_KHW_Servo_setValue.rAux[1], sv_rDrivePressure);
b := WRITE_SVREAL_DIRECT(sv_KHW_Servo_setValue.rVeloc, sv_rDriveVelocity);

@SaTrans 0
@SaExits 0
@END_SfcBody

@@@BEG_Comment@@@
@TL(0)

@@@END_Comment@@@

@BEG_Body
@TL(29)
(**************************************** WARNING ********************************************
 *** The KEBA Kemro K2 System including software is not intended for safety control tasks! ***
 ***                       For further information see Comment tab!                        ***
 *********************************************************************************************)

IF mbInitDone THEN

   IF NOT sv_Servo.ServoState.bError THEN

      //Bit 0: first or second parameter set (first parameter set should be default)
      //Bit 1: master or slave (master = 0, slave = 1)
      IF bMaster THEN
         rTmp := 0.0;
      ELSE
         rTmp := 2.0;
      END_IF;

      IF CHECK_REF(piCtrlParamSet^) AND (piCtrlParamSet^ = 2) THEN
         rTmp := rTmp + 1.0;
      END_IF;

      b := WRITE_SV_DIRECT(sv_KHW_Servo_setValue.rAux[2], rTmp);

      mbStop := FALSE;
      START_PROCESS_ALGORITHM(paOut);

    END_IF;
END_IF;

@END_Body

@@@BEG_Comment@@@
@TL(0)

@@@END_Comment@@@

@BEG_Body
@TL(7)
(**************************************** WARNING ********************************************
 *** The KEBA Kemro K2 System including software is not intended for safety control tasks! ***
 ***                       For further information see Comment tab!                        ***
 *********************************************************************************************)

mbStop := TRUE;

@END_Body

@@@BEG_Comment@@@
@TL(0)

@@@END_Comment@@@

@BEG_Body
@TL(11)
(**************************************** WARNING ********************************************
 *** The KEBA Kemro K2 System including software is not intended for safety control tasks! ***
 ***                       For further information see Comment tab!                        ***
 *********************************************************************************************)

IF NOT IS_LINKED(sv_KHW_Servo_setValue) THEN
   RETURN;
END_IF;

mbDriveError := sv_Servo.ServoState.bError;

@END_Body

@@@BEG_Comment@@@
@TL(0)

@@@END_Comment@@@

@BEG_Body
@TL(17)
(**************************************** WARNING ********************************************
 *** The KEBA Kemro K2 System including software is not intended for safety control tasks! ***
 ***                       For further information see Comment tab!                        ***
 *********************************************************************************************)

//Force PQ endpoints
IF sv_ForceP.bForce OR sv_ForceQ.bForce THEN
   IF NOT mbForceStarted THEN
      mbForceStarted := TRUE;
      START_PROCESS_ALGORITHM(paPQForce);
   END_IF;
END_IF;

@END_Body

@@@BEG_Comment@@@
@TL(0)

@@@END_Comment@@@

@BEG_Body
@TL(29)
(**************************************** WARNING ********************************************
 *** The KEBA Kemro K2 System including software is not intended for safety control tasks! ***
 ***                       For further information see Comment tab!                        ***
 *********************************************************************************************)

//Force PQ endpoints
IF sv_ForceP.bForce THEN
   rForceP := sv_ForceP.rForceValue / rMaxPressure * 1000.0;
   b := WRITE_SVREAL_DIRECT(sv_KHW_Servo_setValue.rAux[1], rForceP);
   b := WRITE_SVREAL_DIRECT(sv_ForceP.rActualValue, sv_ForceP.rForceValue);
ELSIF NOT sv_ForceP.bForce THEN
   b := WRITE_SVREAL_DIRECT(sv_KHW_Servo_setValue.rAux[1], 0.0);
   b := WRITE_SVREAL_DIRECT(sv_ForceP.rActualValue, 0.0);
END_IF;

IF sv_ForceQ.bForce THEN
   rForceQ := sv_ForceQ.rForceValue * 10.0;
   b := WRITE_SVREAL_DIRECT(sv_KHW_Servo_setValue.rVeloc, rForceQ);
   b := WRITE_SVREAL_DIRECT(sv_ForceQ.rActualValue, sv_ForceQ.rForceValue);
ELSIF NOT sv_ForceQ.bForce THEN
   b := WRITE_SVREAL_DIRECT(sv_KHW_Servo_setValue.rVeloc, 0.0);
   b := WRITE_SVREAL_DIRECT(sv_ForceQ.rActualValue, 0.0);
END_IF;

IF NOT sv_ForceQ.bForce AND NOT sv_ForceP.bForce THEN
   mbForceStarted := FALSE;
   STOP_PROCESS_ALGORITHM();
END_IF;

@END_Body

@@@BEG_Comment@@@
@TL(0)

@@@END_Comment@@@
@END_Body

@END_Contents

(* ---- ABPumpControl.pu ---- *)
(*
@h    ! WARNING !
@h    The Kemro K2 system (including software) only meets category B according to EN 954-1,
@h    thus it is not intended for usage in safety-relevant control applications in the field
@h    of personal safety (e.g. emergency stop).
@h    To implement potentially necessary safety-relevant control tasks, always use additional
@h    external safety devices that are intended for the particular purpose, and meet the necessary
@h    functional safety.
@h    For further information see EN 954-1 (EN ISO 13849-1) and/or the K2-x00 user manual, chapter
@h    "CE conformity, directives and standards".

This AB controls the analog output to a pump.
Depending on the evAnaDevCmd events (sent by outputcoordination), the output blocks are started or stopped.
The response event (evAnaDevResponse) is sent after the output block is stopped (nAnaDevStopped).

Attention!!
It is not allowed to send response events without receiving an according nAnaDevCmd event before.

*)

IMPORT_OVER_LISTFILE
 GET_SYNC_REFTO
, SET_EVENT
, tevAnaDevCmd
, tsDeviceId
, KAPPL_LintabData
, ABPumpOutput
, tevAnaDevResponse
, tevAnaDevResponseData
, tyPumpData
, tyCalibDevices
, KSYS_Status
, tevAnaDevCmdData

END_IMPORT

ALGORITHM_BLOCK ABPumpControl #DUMMY_EDIT_BLOCK

SYSTEM_VAR
 sv_DeviceId : tsDeviceId;
 sv_rPressure : REAL;
 sv_rVelocity : REAL;
 sv_rAbsFlow : REAL;
 sv_VelocityLintab : KAPPL_LintabData;
 sv_PressureLintab : KAPPL_LintabData;
 sv_VelocityLintabPVCalib : KAPPL_LintabData (* lintab for pump PV calib -> to directly output voltage *);
 sv_PressureLintabPVCalib : KAPPL_LintabData (* lintab for pump PV calib -> to directly output voltage *);
 sv_iPumpFlowChanged : DINT (* must be increased by every pump if sv_rAbsFlow is changed *);
 sv_rMaxPressure : REAL;
 sv_iPumpPressureChanged : DINT (* must be increased by every pump if sv_rMaxPressure is changed *);
 ao_Pressure : REAL;
 ao_Velocity : REAL;
 sv_PumpData : tyPumpData;
 sv_PumpCalibDevices : tyCalibDevices (* !!! device 1 - 20 reserved !!! *);
 sv_iDeviceForCalib : DINT (* index in sv_PumpCalibDevices - list *);
 sv_bDoPumpPressureCalib : BOOL;
 sv_bDoPumpVelocityCalib : BOOL;
 sv_iCalibratingPump : DINT (* number of pump which is actually calibrating *);
 sv_rMaximumPressure : REAL;
 sv_rActPressureHydr : REAL (* actual pressure in bar (measured by pressure sensor) *);
 ai_SysPressure : REAL;
 sv_bDeviceReady : BOOL;
 sv_rMaxVoltagePressure : REAL;
 sv_rMaxVoltageVelocity : REAL;
 sv_rMaxVoltagePressOutput : REAL;
 sv_rMaxVoltageVelOutput : REAL;
END_VAR

SYSTEM_OBJECT
 evAnaDevCmd : tevAnaDevCmd;
 EV_Task_1 : TASK;
 TaskMid : TASK;
 evAnaDevResponse : tevAnaDevResponse;
 PU_Task_7 : TASK;
 TaskInject : TASK;
END_OBJECT

VAR
 abPumpOutput : ABPumpOutput;
 mbStop : BOOL;
 evAnaDevResponseData : tevAnaDevResponseData;
 mprMaxPressure : REFTO REAL;
 mprMaxVoltagePress : REFTO REAL;
 mprMaxVoltageVel : REFTO REAL;
END_VAR

PROCESS_ALGORITHM paInit ON TaskMid AUTOSTART

VAR
 prSysPressure : REFTO REAL;
 s : KSYS_Status;
END_VAR
#BEGIN_EDIT_BLOCK
(**************************************** WARNING ********************************************
 *** The KEBA Kemro K2 System including software is not intended for safety control tasks! ***
 ***                       For further information see Comment tab!                        ***
 *********************************************************************************************)

//write information to sv_PumpData
IF sv_DeviceId.IndexId <= cMaxNrOfPumps THEN
   sv_PumpData[sv_DeviceId.IndexId].prAbsFlow := @sv_rAbsFlow;
   sv_PumpData[sv_DeviceId.IndexId].prAnaOutP := @sv_rPressure;
   sv_PumpData[sv_DeviceId.IndexId].prAnaOutV := @sv_rVelocity;

   //compatibility:
   //use sv_rMaximumPressure for first pump
   //use Injection1.ai_SysPressure for actual system pressure of first pump
   IF sv_DeviceId.IndexId = 1 THEN
      sv_PumpData[sv_DeviceId.IndexId].prMaxPressure := @sv_rMaximumPressure;
      prSysPressure := GET_SYNC_REFTO("Injection1.ai_SysPressure", T#0s, s);
      IF s = KSYS_Status_OK THEN
         prSysPressure := GET_SYNC_REFTO("Injection1.sv_rActSysPressure", T#0s, s);
         sv_PumpData[sv_DeviceId.IndexId].prActSysPressure := prSysPressure;
      END_IF;
      mprMaxVoltagePress := @sv_rMaxVoltagePressure;
      mprMaxVoltageVel := @sv_rMaxVoltageVelocity;
   ELSE
      sv_PumpData[sv_DeviceId.IndexId].prMaxPressure := @sv_rMaxPressure;
      IF IS_LINKED(ai_SysPressure) THEN
         sv_PumpData[sv_DeviceId.IndexId].prActSysPressure := @sv_rActPressureHydr;
      END_IF;
   END_IF;

   sv_PumpData[sv_DeviceId.IndexId].prActVoltageP := @ao_Pressure;
   sv_PumpData[sv_DeviceId.IndexId].prActVoltageV := @ao_Velocity;
   sv_PumpData[sv_DeviceId.IndexId].prMaxVoltageP := @sv_rMaxVoltagePressOutput;
   sv_PumpData[sv_DeviceId.IndexId].prMaxVoltageV := @sv_rMaxVoltageVelOutput;

   mprMaxPressure := sv_PumpData[sv_DeviceId.IndexId].prMaxPressure;
END_IF;

STOP_PROCESS_ALGORITHM();

;#END_EDIT_BLOCK END_ALGORITHM

EVENT_ALGORITHM evaAnaDevCmd ON EV_Task_1 WITH evAnaDevCmd

VAR_INPUT
 evAnaDevCmdData : tevAnaDevCmdData;
END_VAR

VAR
 bPumpCalibActive : BOOL;
END_VAR
#BEGIN_EDIT_BLOCK
(**************************************** WARNING ********************************************
 *** The KEBA Kemro K2 System including software is not intended for safety control tasks! ***
 ***                       For further information see Comment tab!                        ***
 *********************************************************************************************)

IF evAnaDevCmdData.DeviceId = sv_DeviceId THEN
(* received command from OutputCoordination *)
    CASE evAnaDevCmdData.Cmd OF

       nAnaDevStart:    // start pump output
                        mbStop := FALSE;

                        bPumpCalibActive := FALSE;
                        IF sv_iCalibratingPump = sv_DeviceId.IndexId THEN
                           IF ((sv_bDoPumpVelocityCalib AND evAnaDevCmdData.MoveId = sv_PumpCalibDevices[sv_iDeviceForCalib].pVelCalibMovement^.MoveId) OR
                              (sv_bDoPumpPressureCalib AND evAnaDevCmdData.MoveId = sv_PumpCalibDevices[sv_iDeviceForCalib].pPresCalibMovement^.MoveId)) THEN
                              bPumpCalibActive := TRUE;
                           END_IF;
                        END_IF;

                        IF bPumpCalibActive OR evAnaDevCmdData.MoveId = cMoveServoCalib THEN
                           abPumpOutput.aStart.pLintabP := @sv_PressureLintabPVCalib;
                           abPumpOutput.aStart.pLintabV := @sv_VelocityLintabPVCalib;
                        ELSE
                           abPumpOutput.aStart.pLintabP := @sv_PressureLintab;
                           abPumpOutput.aStart.pLintabV := @sv_VelocityLintab;
                        END_IF;

                        abPumpOutput.aStart(AnaOutMode := evAnaDevCmdData.Mode,
                                            prPressure := evAnaDevCmdData.prAnaOutP,
                                            prVelocity := evAnaDevCmdData.prAnaOutV);

                        sv_bDeviceReady := FALSE;

                        START_PROCESS_ALGORITHM(paRun);

       nAnaDevStop:     // stop pump output
                        mbStop := TRUE;

    END_CASE;
END_IF;

;#END_EDIT_BLOCK END_ALGORITHM

PROCESS_ALGORITHM paRun ON TaskInject AUTOSTART

(* IecGraph-Code *)

(* init step *)
INITIAL_STEP INIT:
END_STEP

(* steps *)
STEP WAIT_FOR_STOP_CMD:
END_STEP

STEP STOP_OUTPUT:
AStop (N);
END_STEP

ACTION AStop: #BEGIN_EDIT_BLOCK
(* Stopping Pump Output *)
abPumpOutput.aStop();

;#END_EDIT_BLOCK END_ACTION (*AStop*)
STEP STOPPED:
AStopped (P);
END_STEP

ACTION AStopped: #BEGIN_EDIT_BLOCK
STOP_PROCESS_ALGORITHM();
// send response to OutputCoordination
evAnaDevResponseData.DeviceId := sv_DeviceId;
evAnaDevResponseData.State := nAnaDevStopped;
SET_EVENT(evAnaDevResponse, evAnaDevResponseData);

sv_bDeviceReady := TRUE;

;#END_EDIT_BLOCK END_ACTION (*AStopped*)

(* transitions *)
GO_ON_TRANSITION Trans1 (* Trans1 *) FROM INIT TO WAIT_FOR_STOP_CMD :=  #BEGIN_EDIT_BLOCK
TRUE
;#END_EDIT_BLOCK
END_TRANSITION

GO_ON_TRANSITION TStopCmdReceived (* Trans2 *) FROM WAIT_FOR_STOP_CMD TO STOP_OUTPUT :=  #BEGIN_EDIT_BLOCK
mbStop
;#END_EDIT_BLOCK
END_TRANSITION

GO_ON_TRANSITION TOutputStopped (* Trans7 *) FROM STOP_OUTPUT TO STOPPED :=  #BEGIN_EDIT_BLOCK
abPumpOutput.aStop.bReady
;#END_EDIT_BLOCK
END_TRANSITION

TRANSITION Trans3 (* Trans3 *) FROM STOPPED TO WAIT_FOR_STOP_CMD :=  #BEGIN_EDIT_BLOCK
TRUE
;#END_EDIT_BLOCK
END_TRANSITION

(* end IecGraph-Code *)
(* sfc-code *)
(* end sfc-code *)

END_ALGORITHM

POSTUPDATE_ALGORITHM pAbsFlowChanged ON PU_Task_7 WITH sv_rAbsFlow

#BEGIN_EDIT_BLOCK
(**************************************** WARNING ********************************************
 *** The KEBA Kemro K2 System including software is not intended for safety control tasks! ***
 ***                       For further information see Comment tab!                        ***
 *********************************************************************************************)

sv_iPumpFlowChanged := sv_iPumpFlowChanged + 1;

;#END_EDIT_BLOCK END_ALGORITHM

POSTUPDATE_ALGORITHM pMaxPressureChanged ON PU_Task_7 WITH mprMaxPressure^

#BEGIN_EDIT_BLOCK
(**************************************** WARNING ********************************************
 *** The KEBA Kemro K2 System including software is not intended for safety control tasks! ***
 ***                       For further information see Comment tab!                        ***
 *********************************************************************************************)

sv_iPumpPressureChanged := sv_iPumpPressureChanged + 1;

IF (sv_DeviceId.IndexId = 1) THEN
   //only for pump1: copy new maximum pressure to Pump1.sv_rMaxPressure
   //because otherwise some plausibilities are not ok
   sv_rMaxPressure := sv_rMaximumPressure;
END_IF;

;#END_EDIT_BLOCK END_ALGORITHM

POSTUPDATE_ALGORITHM pMaxOutputVoltage ON PU_Task_7 WITH mprMaxVoltagePress^,mprMaxVoltageVel^

#BEGIN_EDIT_BLOCK
(**************************************** WARNING ********************************************
 *** The KEBA Kemro K2 System including software is not intended for safety control tasks! ***
 ***                       For further information see Comment tab!                        ***
 *********************************************************************************************)

//this code is only necessary for pump1 (due to compatibility reasons)
sv_rMaxVoltagePressOutput := mprMaxVoltagePress^;
sv_rMaxVoltageVelOutput := mprMaxVoltageVel^

;#END_EDIT_BLOCK END_ALGORITHM

END_ALGORITHM_BLOCK

#END_OF_IEC_PART

@Puma @IecEditor 6 97 @Pou 25
@@@BEG_Comment@@@
@h    ! WARNING !
@h    The Kemro K2 system (including software) only meets category B according to EN 954-1,
@h    thus it is not intended for usage in safety-relevant control applications in the field
@h    of personal safety (e.g. emergency stop).
@h    To implement potentially necessary safety-relevant control tasks, always use additional
@h    external safety devices that are intended for the particular purpose, and meet the necessary
@h    functional safety.
@h    For further information see EN 954-1 (EN ISO 13849-1) and/or the K2-x00 user manual, chapter
@h    "CE conformity, directives and standards".

This AB controls the analog output to a pump.
Depending on the evAnaDevCmd events (sent by outputcoordination), the output blocks are started or stopped.
The response event (evAnaDevResponse) is sent after the output block is stopped (nAnaDevStopped).

Attention!!
It is not allowed to send response events without receiving an according nAnaDevCmd event before.

@@@END_Comment@@@

@BEG_Contents

@BEG_Func
@RT(17)FuncTreeContainer
2
@Var @RT(14)GET_SYNC_REFTO @RT(0) @T @T @DERIVED 0 @F @RT(22)KEBA_STANDARD_FUNCTION @F
@T
@BEG_Attrib
0 @RT(0) @RT(0)
@END_Attrib
1 1 @F @F @F @F

@Var @RT(9)SET_EVENT @RT(0) @T @T @DERIVED 0 @F @RT(23)KEBA_STANDARD_PROCEDURE @F
@T
@BEG_Attrib
0 @RT(0) @RT(0)
@END_Attrib
1 1 @F @F @F @F

@END_Func

@BEG_Const
@RT(18)ConstTreeContainer
0
@END_Const

@BEG_Export

@BEG_Kind
@ALGORITHM_BLOCK @RT(13)ABPumpControl @STRUCTURED_TEXT
@RT(0) @RT(0) @RT(0)
@END_Kind

@BEG_Dcl
@RT(16)DclTreeContainer
39
@Var @RT(11)evAnaDevCmd @RT(0) @T @T @DERIVED 0 @T @T @DT @RT(12)tevAnaDevCmd @RT(0) @T @T @UNKNOWN 0 @F
@F @F
@T
@BEG_Attrib
3 @RT(0) @RT(0) @RT(0)
@END_Attrib
1 7 @F @F @F @F

@Var @RT(9)EV_Task_1 @RT(0) @T @T @RENAMED 0 @T @T @DT @RT(4)TASK @RT(0) @T @T @BASIC 0 @F
@F @F
@T
@BEG_Attrib
3 @RT(0) @RT(0) @RT(0)
@END_Attrib
1 7 @F @F @F @F

@Var @RT(11)sv_DeviceId @RT(0) @T @T @DERIVED 0 @T @T @DT @RT(10)tsDeviceId @RT(0) @T @T @UNKNOWN 0 @F
@F @F
@T
@BEG_Attrib
3 @RT(0) @RT(0) @RT(0)
@END_Attrib
1 8 @F @F @F @F

@Var @RT(12)sv_rPressure @RT(0) @T @F @DT @RT(4)REAL @RT(0) @T @T @BASIC 0 @F
@F @F
@T
@BEG_Attrib
3 @RT(0) @RT(0) @RT(0)
@END_Attrib
1 8 @F @F @F @F

@Var @RT(12)sv_rVelocity @RT(0) @T @F @DT @RT(4)REAL @RT(0) @T @T @BASIC 0 @F
@F @F
@T
@BEG_Attrib
3 @RT(0) @RT(0) @RT(0)
@END_Attrib
1 8 @F @F @F @F

@Var @RT(11)sv_rAbsFlow @RT(0) @T @F @DT @RT(4)REAL @RT(0) @T @T @BASIC 0 @F
@F @F
@T
@BEG_Attrib
3 @RT(0) @RT(0) @RT(0)
@END_Attrib
1 8 @F @F @F @F

@Var @RT(17)sv_VelocityLintab @RT(0) @T @T @DERIVED 0 @T @T @DT @RT(16)KAPPL_LintabData @RT(0) @T @T @UNKNOWN 0 @F
@F @F
@T
@BEG_Attrib
3 @RT(0) @RT(0) @RT(0)
@END_Attrib
1 8 @F @F @F @F

@Var @RT(17)sv_PressureLintab @RT(0) @T @T @DERIVED 0 @T @T @DT @RT(16)KAPPL_LintabData @RT(0) @T @T @UNKNOWN 0 @F
@F @F
@T
@BEG_Attrib
3 @RT(0) @RT(0) @RT(0)
@END_Attrib
1 8 @F @F @F @F

@Var @RT(12)abPumpOutput @RT(0) @T @T @DERIVED 0 @T @T @DT @RT(12)ABPumpOutput @RT(0) @T @T @UNKNOWN 0 @F
@F @F
@T
@BEG_Attrib
3 @RT(0) @RT(0) @RT(0)
@END_Attrib
1 0 @F @F @F @F

@Var @RT(7)TaskMid @RT(0) @T @T @RENAMED 0 @T @T @DT @RT(4)TASK @RT(0) @T @T @BASIC 0 @F
@F @F
@T
@BEG_Attrib
3 @RT(0) @RT(0) @RT(0)
@END_Attrib
1 7 @F @F @F @F

@Var @RT(6)mbStop @RT(0) @T @F @DT @RT(4)BOOL @RT(0) @T @T @BASIC 0 @F
@F @F
@T
@BEG_Attrib
3 @RT(0) @RT(0) @RT(0)
@END_Attrib
1 0 @F @F @F @F

@Var @RT(16)evAnaDevResponse @RT(0) @T @T @DERIVED 0 @T @T @DT @RT(17)tevAnaDevResponse @RT(0) @T @T @UNKNOWN 0 @F
@F @F
@T
@BEG_Attrib
3 @RT(0) @RT(0) @RT(0)
@END_Attrib
1 7 @F @F @F @F

@Var @RT(20)evAnaDevResponseData @RT(0) @T @T @DERIVED 0 @T @T @DT @RT(21)tevAnaDevResponseData @RT(0) @T @T @UNKNOWN 0 @F
@F @F
@T
@BEG_Attrib
3 @RT(0) @RT(0) @RT(0)
@END_Attrib
1 0 @F @F @F @F

@Var @RT(24)sv_VelocityLintabPVCalib @RT(0) @T @T @DERIVED 0 @T @T @DT @RT(16)KAPPL_LintabData @RT(0) @T @T @UNKNOWN 0 @F
@F @F
@T
@BEG_Attrib
3 @RT(0) @RT(54)lintab for pump PV calib -> to directly output voltage @RT(0)
@END_Attrib
1 8 @F @F @F @F

@Var @RT(24)sv_PressureLintabPVCalib @RT(0) @T @T @DERIVED 0 @T @T @DT @RT(16)KAPPL_LintabData @RT(0) @T @T @UNKNOWN 0 @F
@F @F
@T
@BEG_Attrib
3 @RT(0) @RT(54)lintab for pump PV calib -> to directly output voltage @RT(0)
@END_Attrib
1 8 @F @F @F @F

@Var @RT(9)PU_Task_7 @RT(0) @T @T @RENAMED 0 @T @T @DT @RT(4)TASK @RT(0) @T @T @BASIC 0 @F
@F @F
@T
@BEG_Attrib
3 @RT(0) @RT(0) @RT(0)
@END_Attrib
1 7 @F @F @F @F

@Var @RT(19)sv_iPumpFlowChanged @RT(0) @T @F @DT @RT(4)DINT @RT(0) @T @T @BASIC 0 @F
@F @F
@T
@BEG_Attrib
3 @RT(0) @RT(57)must be increased by every pump if sv_rAbsFlow is changed @RT(0)
@END_Attrib
1 8 @F @F @F @F

@Var @RT(15)sv_rMaxPressure @RT(0) @T @F @DT @RT(4)REAL @RT(0) @T @T @BASIC 0 @F
@F @F
@T
@BEG_Attrib
3 @RT(0) @RT(0) @RT(0)
@END_Attrib
1 8 @F @F @F @F

@Var @RT(23)sv_iPumpPressureChanged @RT(0) @T @F @DT @RT(4)DINT @RT(0) @T @T @BASIC 0 @F
@F @F
@T
@BEG_Attrib
3 @RT(0) @RT(61)must be increased by every pump if sv_rMaxPressure is changed @RT(0)
@END_Attrib
1 8 @F @F @F @F

@Var @RT(11)ao_Pressure @RT(0) @T @F @DT @RT(4)REAL @RT(0) @T @T @BASIC 0 @F
@F @F
@T
@BEG_Attrib
3 @RT(0) @RT(0) @RT(0)
@END_Attrib
1 8 @F @F @F @F

@Var @RT(11)ao_Velocity @RT(0) @T @F @DT @RT(4)REAL @RT(0) @T @T @BASIC 0 @F
@F @F
@T
@BEG_Attrib
3 @RT(0) @RT(0) @RT(0)
@END_Attrib
1 8 @F @F @F @F

@Var @RT(11)sv_PumpData @RT(0) @T @T @DERIVED 0 @T @T @DT @RT(10)tyPumpData @RT(0) @T @T @UNKNOWN 0 @F
@F @F
@T
@BEG_Attrib
3 @RT(0) @RT(0) @RT(0)
@END_Attrib
1 8 @F @F @F @F

@Var @RT(19)sv_PumpCalibDevices @RT(0) @T @T @DERIVED 0 @T @T @DT @RT(14)tyCalibDevices @RT(0) @T @T @UNKNOWN 0 @F
@F @F
@T
@BEG_Attrib
3 @RT(0) @RT(30)!!! device 1 - 20 reserved !!! @RT(0)
@END_Attrib
1 8 @F @F @F @F

@Var @RT(18)sv_iDeviceForCalib @RT(0) @T @F @DT @RT(4)DINT @RT(0) @T @T @BASIC 0 @F
@F @F
@T
@BEG_Attrib
3 @RT(0) @RT(35)index in sv_PumpCalibDevices - list @RT(0)
@END_Attrib
1 8 @F @F @F @F

@Var @RT(23)sv_bDoPumpPressureCalib @RT(0) @T @F @DT @RT(4)BOOL @RT(0) @T @T @BASIC 0 @F
@F @F
@T
@BEG_Attrib
3 @RT(0) @RT(0) @RT(0)
@END_Attrib
1 8 @F @F @F @F

@Var @RT(23)sv_bDoPumpVelocityCalib @RT(0) @T @F @DT @RT(4)BOOL @RT(0) @T @T @BASIC 0 @F
@F @F
@T
@BEG_Attrib
3 @RT(0) @RT(0) @RT(0)
@END_Attrib
1 8 @F @F @F @F

@Var @RT(19)sv_iCalibratingPump @RT(0) @T @F @DT @RT(4)DINT @RT(0) @T @T @BASIC 0 @F
@F @F
@T
@BEG_Attrib
3 @RT(0) @RT(44)number of pump which is actually calibrating @RT(0)
@END_Attrib
1 8 @F @F @F @F

@Var @RT(19)sv_rMaximumPressure @RT(0) @T @F @DT @RT(4)REAL @RT(0) @T @T @BASIC 0 @F
@F @F
@T
@BEG_Attrib
3 @RT(0) @RT(0) @RT(0)
@END_Attrib
1 8 @F @F @F @F

@Var @RT(14)mprMaxPressure @RT(0) @T @T @REFTO 0 @T @DT @RT(4)REAL @RT(0) @T @T @BASIC 0 @F
@F @F
@T
@BEG_Attrib
3 @RT(0) @RT(0) @RT(0)
@END_Attrib
1 0 @F @F @F @F

@Var @RT(19)sv_rActPressureHydr @RT(0) @T @F @DT @RT(4)REAL @RT(0) @T @T @BASIC 0 @F
@F @F
@T
@BEG_Attrib
3 @RT(0) @RT(52)actual pressure in bar (measured by pressure sensor) @RT(0)
@END_Attrib
1 8 @F @F @F @F

@Var @RT(14)ai_SysPressure @RT(0) @T @F @DT @RT(4)REAL @RT(0) @T @T @BASIC 0 @F
@F @F
@T
@BEG_Attrib
3 @RT(0) @RT(0) @RT(0)
@END_Attrib
1 8 @F @F @F @F

@Var @RT(15)sv_bDeviceReady @RT(0) @T @F @DT @RT(4)BOOL @RT(0) @T @T @BASIC 0 @F
@F @F
@T
@BEG_Attrib
3 @RT(0) @RT(0) @RT(0)
@END_Attrib
1 8 @F @F @F @F

@Var @RT(10)TaskInject @RT(0) @T @T @RENAMED 0 @T @T @DT @RT(4)TASK @RT(0) @T @T @BASIC 0 @F
@F @F
@T
@BEG_Attrib
3 @RT(0) @RT(0) @RT(0)
@END_Attrib
1 7 @F @F @F @F

@Var @RT(22)sv_rMaxVoltagePressure @RT(0) @T @F @DT @RT(4)REAL @RT(0) @T @T @BASIC 0 @F
@F @F
@T
@BEG_Attrib
3 @RT(0) @RT(0) @RT(0)
@END_Attrib
1 8 @F @F @F @F

@Var @RT(22)sv_rMaxVoltageVelocity @RT(0) @T @F @DT @RT(4)REAL @RT(0) @T @T @BASIC 0 @F
@F @F
@T
@BEG_Attrib
3 @RT(0) @RT(0) @RT(0)
@END_Attrib
1 8 @F @F @F @F

@Var @RT(25)sv_rMaxVoltagePressOutput @RT(0) @T @F @DT @RT(4)REAL @RT(0) @T @T @BASIC 0 @F
@F @F
@T
@BEG_Attrib
3 @RT(0) @RT(0) @RT(0)
@END_Attrib
1 8 @F @F @F @F

@Var @RT(23)sv_rMaxVoltageVelOutput @RT(0) @T @F @DT @RT(4)REAL @RT(0) @T @T @BASIC 0 @F
@F @F
@T
@BEG_Attrib
3 @RT(0) @RT(0) @RT(0)
@END_Attrib
1 8 @F @F @F @F

@Var @RT(18)mprMaxVoltagePress @RT(0) @T @T @REFTO 0 @T @DT @RT(4)REAL @RT(0) @T @T @BASIC 0 @F
@F @F
@T
@BEG_Attrib
3 @RT(0) @RT(0) @RT(0)
@END_Attrib
1 0 @F @F @F @F

@Var @RT(16)mprMaxVoltageVel @RT(0) @T @T @REFTO 0 @T @DT @RT(4)REAL @RT(0) @T @T @BASIC 0 @F
@F @F
@T
@BEG_Attrib
3 @RT(0) @RT(0) @RT(0)
@END_Attrib
1 0 @F @F @F @F

@END_Dcl

@END_Export

@BEG_Body

6

@BEG_Export

@BEG_Algo
@PROCESS_ALGORITHM @RT(6)paInit @STRUCTURED_TEXT
@RT(0) @RT(0) @RT(7)TaskMid @T @F
@END_Algo

@BEG_Dcl
@RT(16)DclTreeContainer
2
@Var @RT(13)prSysPressure @RT(0) @T @T @REFTO 0 @T @DT @RT(4)REAL @RT(0) @T @T @BASIC 0 @F
@F @F
@T
@BEG_Attrib
3 @RT(0) @RT(0) @RT(0)
@END_Attrib
1 0 @F @F @F @F

@Var @RT(1)s @RT(0) @T @T @DERIVED 0 @T @T @DT @RT(11)KSYS_Status @RT(0) @T @T @UNKNOWN 0 @F
@F @F
@T
@BEG_Attrib
3 @RT(0) @RT(0) @RT(0)
@END_Attrib
1 0 @F @F @F @F

@END_Dcl

@END_Export

@BEG_Export

@BEG_Algo
@EVENT_ALGORITHM @RT(12)evaAnaDevCmd @STRUCTURED_TEXT
@RT(0) @RT(11)evAnaDevCmd @RT(9)EV_Task_1 @F @F
@END_Algo

@BEG_Dcl
@RT(16)DclTreeContainer
2
@Var @RT(15)evAnaDevCmdData @RT(0) @T @T @DERIVED 0 @T @T @DT @RT(16)tevAnaDevCmdData @RT(0) @T @T @UNKNOWN 0 @F
@F @F
@T
@BEG_Attrib
3 @RT(0) @RT(0) @RT(0)
@END_Attrib
1 1 @F @F @F @F

@Var @RT(16)bPumpCalibActive @RT(0) @T @F @DT @RT(4)BOOL @RT(0) @T @T @BASIC 0 @F
@F @F
@T
@BEG_Attrib
3 @RT(0) @RT(0) @RT(0)
@END_Attrib
1 0 @F @F @F @F

@END_Dcl

@END_Export

@BEG_Export

@BEG_Algo
@PROCESS_ALGORITHM @RT(5)paRun @SEQUENTIAL_FLOW_CHART
@RT(0) @RT(0) @RT(10)TaskInject @T @F
@END_Algo

@BEG_Dcl
@RT(16)DclTreeContainer
0
@END_Dcl

@END_Export

@BEG_Export

@BEG_Algo
@POSTUPDATE_ALGORITHM @RT(15)pAbsFlowChanged @STRUCTURED_TEXT
@RT(0) @RT(11)sv_rAbsFlow @RT(9)PU_Task_7 @F @F
@END_Algo

@BEG_Dcl
@RT(16)DclTreeContainer
0
@END_Dcl

@END_Export

@BEG_Export

@BEG_Algo
@POSTUPDATE_ALGORITHM @RT(19)pMaxPressureChanged @STRUCTURED_TEXT
@RT(0) @RT(15)mprMaxPressure^ @RT(9)PU_Task_7 @F @F
@END_Algo

@BEG_Dcl
@RT(16)DclTreeContainer
0
@END_Dcl

@END_Export

@BEG_Export

@BEG_Algo
@POSTUPDATE_ALGORITHM @RT(17)pMaxOutputVoltage @STRUCTURED_TEXT
@RT(0) @RT(37)mprMaxVoltagePress^,mprMaxVoltageVel^ @RT(9)PU_Task_7 @F @F
@END_Algo

@BEG_Dcl
@RT(16)DclTreeContainer
0
@END_Dcl

@END_Export

@BEG_Body
@TL(40)
(**************************************** WARNING ********************************************
 *** The KEBA Kemro K2 System including software is not intended for safety control tasks! ***
 ***                       For further information see Comment tab!                        ***
 *********************************************************************************************)

//write information to sv_PumpData
IF sv_DeviceId.IndexId <= cMaxNrOfPumps THEN
   sv_PumpData[sv_DeviceId.IndexId].prAbsFlow := @sv_rAbsFlow;
   sv_PumpData[sv_DeviceId.IndexId].prAnaOutP := @sv_rPressure;
   sv_PumpData[sv_DeviceId.IndexId].prAnaOutV := @sv_rVelocity;

   //compatibility:
   //use sv_rMaximumPressure for first pump
   //use Injection1.ai_SysPressure for actual system pressure of first pump
   IF sv_DeviceId.IndexId = 1 THEN
      sv_PumpData[sv_DeviceId.IndexId].prMaxPressure := @sv_rMaximumPressure;
      prSysPressure := GET_SYNC_REFTO("Injection1.ai_SysPressure", T#0s, s);
      IF s = KSYS_Status_OK THEN
         prSysPressure := GET_SYNC_REFTO("Injection1.sv_rActSysPressure", T#0s, s);
         sv_PumpData[sv_DeviceId.IndexId].prActSysPressure := prSysPressure;
      END_IF;
      mprMaxVoltagePress := @sv_rMaxVoltagePressure;
      mprMaxVoltageVel := @sv_rMaxVoltageVelocity;
   ELSE
      sv_PumpData[sv_DeviceId.IndexId].prMaxPressure := @sv_rMaxPressure;
      IF IS_LINKED(ai_SysPressure) THEN
         sv_PumpData[sv_DeviceId.IndexId].prActSysPressure := @sv_rActPressureHydr;
      END_IF;
   END_IF;

   sv_PumpData[sv_DeviceId.IndexId].prActVoltageP := @ao_Pressure;
   sv_PumpData[sv_DeviceId.IndexId].prActVoltageV := @ao_Velocity;
   sv_PumpData[sv_DeviceId.IndexId].prMaxVoltageP := @sv_rMaxVoltagePressOutput;
   sv_PumpData[sv_DeviceId.IndexId].prMaxVoltageV := @sv_rMaxVoltageVelOutput;

   mprMaxPressure := sv_PumpData[sv_DeviceId.IndexId].prMaxPressure;
END_IF;

STOP_PROCESS_ALGORITHM();

@END_Body

@@@BEG_Comment@@@
@TL(0)

@@@END_Comment@@@

@BEG_Body
@TL(42)
(**************************************** WARNING ********************************************
 *** The KEBA Kemro K2 System including software is not intended for safety control tasks! ***
 ***                       For further information see Comment tab!                        ***
 *********************************************************************************************)

IF evAnaDevCmdData.DeviceId = sv_DeviceId THEN
(* received command from OutputCoordination *)
    CASE evAnaDevCmdData.Cmd OF

       nAnaDevStart:    // start pump output
                        mbStop := FALSE;

                        bPumpCalibActive := FALSE;
                        IF sv_iCalibratingPump = sv_DeviceId.IndexId THEN
                           IF ((sv_bDoPumpVelocityCalib AND evAnaDevCmdData.MoveId = sv_PumpCalibDevices[sv_iDeviceForCalib].pVelCalibMovement^.MoveId) OR
                              (sv_bDoPumpPressureCalib AND evAnaDevCmdData.MoveId = sv_PumpCalibDevices[sv_iDeviceForCalib].pPresCalibMovement^.MoveId)) THEN
                              bPumpCalibActive := TRUE;
                           END_IF;
                        END_IF;

                        IF bPumpCalibActive OR evAnaDevCmdData.MoveId = cMoveServoCalib THEN
                           abPumpOutput.aStart.pLintabP := @sv_PressureLintabPVCalib;
                           abPumpOutput.aStart.pLintabV := @sv_VelocityLintabPVCalib;
                        ELSE
                           abPumpOutput.aStart.pLintabP := @sv_PressureLintab;
                           abPumpOutput.aStart.pLintabV := @sv_VelocityLintab;
                        END_IF;

                        abPumpOutput.aStart(AnaOutMode := evAnaDevCmdData.Mode,
                                            prPressure := evAnaDevCmdData.prAnaOutP,
                                            prVelocity := evAnaDevCmdData.prAnaOutV);

                        sv_bDeviceReady := FALSE;

                        START_PROCESS_ALGORITHM(paRun);

       nAnaDevStop:     // stop pump output
                        mbStop := TRUE;

    END_CASE;
END_IF;

@END_Body

@@@BEG_Comment@@@
@TL(0)

@@@END_Comment@@@

@BEG_SfcBody
12 8 8

@BEG_SfcData 2
@StepSeq @RT(4)sseq @F 3
@Step @RT(4)INIT @F @T @F @F @RT(0) @F
@AcbCont @RT(7)unnamed @F 0

@Trans @RT(6)Trans1 @F @T @F @F @T @F @TL(2)
TRUE

@RT(6)Trans1 @F
@Loop @RT(4)loop @F 2
@StepSeq @RT(3)seq @F 5
@Step @RT(17)WAIT_FOR_STOP_CMD @F @F @F @F @RT(0) @F
@AcbCont @RT(7)unnamed @F 0

@Trans @RT(16)TStopCmdReceived @F @T @F @F @T @F @TL(2)
mbStop

@RT(6)Trans2 @F
@Step @RT(11)STOP_OUTPUT @F @F @F @F @RT(0) @F
@AcbCont @RT(7)unnamed @F 1
@Acb @RT(5)AStop @F @T @RT(1)N @RT(0) @F @F @T @TL(3)
(* Stopping Pump Output *)
abPumpOutput.aStop();

@F

@Trans @RT(14)TOutputStopped @F @T @F @F @T @F @TL(2)
abPumpOutput.aStop.bReady

@RT(6)Trans7 @F
@Step @RT(7)STOPPED @F @F @F @F @RT(0) @F
@AcbCont @RT(7)unnamed @F 1
@Acb @RT(8)AStopped @F @T @RT(1)P @RT(0) @F @F @T @TL(8)
STOP_PROCESS_ALGORITHM();
// send response to OutputCoordination
evAnaDevResponseData.DeviceId := sv_DeviceId;
evAnaDevResponseData.State := nAnaDevStopped;
SET_EVENT(evAnaDevResponse, evAnaDevResponseData);

sv_bDeviceReady := TRUE;

@F

@Trans @RT(6)Trans3 @F @T @T @T @T @T @TL(2)
TRUE

@RT(6)Trans3 @F

@END_SfcData
@SaActions 0
@SaTrans 0
@SaExits 0
@END_SfcBody

@@@BEG_Comment@@@
@TL(0)

@@@END_Comment@@@

@BEG_Body
@TL(7)
(**************************************** WARNING ********************************************
 *** The KEBA Kemro K2 System including software is not intended for safety control tasks! ***
 ***                       For further information see Comment tab!                        ***
 *********************************************************************************************)

sv_iPumpFlowChanged := sv_iPumpFlowChanged + 1;

@END_Body

@@@BEG_Comment@@@
@TL(0)

@@@END_Comment@@@

@BEG_Body
@TL(13)
(**************************************** WARNING ********************************************
 *** The KEBA Kemro K2 System including software is not intended for safety control tasks! ***
 ***                       For further information see Comment tab!                        ***
 *********************************************************************************************)

sv_iPumpPressureChanged := sv_iPumpPressureChanged + 1;

IF (sv_DeviceId.IndexId = 1) THEN
   //only for pump1: copy new maximum pressure to Pump1.sv_rMaxPressure
   //because otherwise some plausibilities are not ok
   sv_rMaxPressure := sv_rMaximumPressure;
END_IF;

@END_Body

@@@BEG_Comment@@@
@TL(0)

@@@END_Comment@@@

@BEG_Body
@TL(9)
(**************************************** WARNING ********************************************
 *** The KEBA Kemro K2 System including software is not intended for safety control tasks! ***
 ***                       For further information see Comment tab!                        ***
 *********************************************************************************************)

//this code is only necessary for pump1 (due to compatibility reasons)
sv_rMaxVoltagePressOutput := mprMaxVoltagePress^;
sv_rMaxVoltageVelOutput := mprMaxVoltageVel^

@END_Body

@@@BEG_Comment@@@
@TL(0)

@@@END_Comment@@@
@END_Body

@END_Contents
